Staubli VAL3: calcTool4p7En.pjx

--- calcTool4p7En.pjx ---
Parameters version=s7.3.1 stackSize=5000 millimeterUnit=true
Program file=aMainTcp.pgx
Program file=aTcp.pgx
Program file=buildTool.pgx
Program file=calculation.pgx
Program file=description.pgx
Program file=example.pgx
Program file=language.pgx
Program file=readme.pgx
Program file=splitUp.pgx
Program file=start.pgx
Program file=stop.pgx
Program file=teachPoints.pgx
Program file=usrButtonTxt.pgx
Program file=valSetBack.pgx
Data file=calcTool4p7En.dtx

--- calcTool4p7En.dtx ---
bool bAbort = true
num nLangSet = 100
num nS1[4]
num nS2[4]
num nS3[4]
num nS4[4]
num nScX
num nScY
num nScZ
num nToolX = 192.690167
num nToolY = -28.471807
num nToolZ = 149.691768
num nXPosButTxt[9]
  [2] = 5
  [3] = 10
  [4] = 15
  [5] = 20
  [6] = 25
  [7] = 30
  [8] = 35
num nYPosButTxt = 13
pointRx pTempS[5]
  [0] = {fatherId=world[0]}
  [1] = {x=378.320625, y=240.768097, z=466.569838, rx=-127.167365, ry=20.154779, rz=59.793558, shoulder=lefty, elbow=epositive, wrist=wpositive, fatherId=world[0]}
  [2] = {x=378.320625, y=240.768097, z=466.569838, rx=-127.167365, ry=20.154779, rz=59.793558, shoulder=lefty, elbow=epositive, wrist=wpositive, fatherId=world[0]}
  [3] = {x=378.320625, y=240.768097, z=466.569838, rx=-127.167365, ry=20.154779, rz=59.793558, shoulder=lefty, elbow=epositive, wrist=wpositive, fatherId=world[0]}
  [4] = {x=378.320625, y=240.768097, z=466.569838, rx=-127.167365, ry=20.154779, rz=59.793558, shoulder=lefty, elbow=epositive, wrist=wpositive, fatherId=world[0]}
string sUsrMess[140]
  [0] = "Please select a Language"
  [1] = "Programm zur Toolberechnung"
  [2] = "Dieses Prog. errechnet anhand 4 POINTS,"
  [3] = "die kugelfoermig um einen gemeinsamen"
  [4] = "Mittelpkt angeordnet sind,die X, Y und"
  [5] = "Z-Werte des akt. Tools. Diese Points"
  [6] = "muessen geometrisch unabhaengig sein."
  [7] = "D.h. sie duerfen nicht in EINER"
  [8] = "gemeinsamen Ebene liegen !!!"
  [9] = "Teachen der Locations !"
  [10] = "Punkt aufnehmen "
  [11] = "Aufnahme des "
  [12] = ".Punkts"
  [13] = "-Here- druecken um Punkt zu speichern"
  [14] = "ABBRUCH"
  [15] = "VORGANG ABGEBROCHEN !!!"
  [16] = ".Punkt aufgenommen !!!"
  [17] = "Mitte"
  [18] = "gemittelt"
  [19] = "Gemitteltes Tool sofort setzten ?"
  [20] = "TOOL NICHT GESETZT !!!"
  [21] = "TOOL GESETZT !!!"
  [22] = "Abbrechen       "
  [23] = "Wollen Sie fortfahren ? "
  [24] = " JA"
  [25] = "NEIN"
  [26] = "Here"
  [27] = "Ergebnis der Toolberechnung"
  [28] = "Tool-X"
  [29] = "Tool-Y"
  [30] = "Tool-Z"
  [31] = "Gemitteltes Tool => TRSF user_tool"
  [32] = "Division durch 0 nicht moeglich !!!"
  [101] = "Program for ToolCalculation"
  [102] = "Program to calculate the Center of a"
  [103] = "Sphere thoughout 4 POINTS which are"
  [104] = "on the surface of his Sphere. The X-,"
  [105] = "Y- and Z-Toolval. will be calcutated."
  [106] = "These POINTS have to be geometricly"
  [107] = "independant=>POINTS don't have to be"
  [108] = "located in ONE plane!!!"
  [109] = "Teaching of Locations !"
  [110] = "Teaching Location"
  [111] = "Teaching of "
  [112] = ".Point"
  [113] = "To teach the Point press - Here -"
  [114] = "ABORT"
  [115] = "PROGRAM ABORTED !!!"
  [116] = ".Point teached !!!"
  [117] = "Center"
  [118] = "average"
  [119] = "Do you want to SET average Tool now ?"
  [120] = "TOOL NOT SET !!!"
  [121] = "TOOL SET !!!"
  [122] = "Abort"
  [123] = "Do you want to continue ?"
  [124] = "YES"
  [125] = " NO"
  [126] = "Here"
  [127] = "Result of the Toolcalculation"
  [128] = "Tool-X"
  [129] = "Tool-Y"
  [130] = "Tool-Z"
  [131] = "Average Tool => TRSF user_tool"
  [132] = "Division though 0 is not possible !!!"
trsf trCenter
trsf trSphere[4]
trsf trTempTool[4]
public trsf trUserTool

--- aMainTcp.pgx ---
public program aMainTcp(num x_nUserLanguage)
  local bool l_bOk
begin
  //-----------------------------------------------------------------------
  //Header begin
  //Description of program
  //  This program creates your tool from 4 different taught positions.
  //  A wizard will guide you through the steps.
  //
  //Input parameters
  //  num x_nUserLanguage :
  //    role : defines the language of GUI (Graphical User Interface) messages
  //    possible values : 1 or 2 : 1 => Deutsch, 2 => English
  //
  //History
  //  Creation : 07-04-08 - f.Rob
  //Header end
  //-----------------------------------------------------------------------

  //Initializing all parameters (trsf, point...)
  call valSetBack()

  //Displays user title depending on the language defined
  title(sUsrMess[1+nLangSet])
  //Displays user instructions
  call description(l_bOk)
  //-> First program for teach the points, after program for calculate sphere,
  //after calculation of the tool components
  if l_bOk==true
    call teachPoints()
    call splitUp(pTempS[1],pTempS[2],pTempS[3],pTempS[4])
    call calculation(nS1[1],nS2[1],nS3[1],nS4[1],nS1[2],nS2[2],nS3[2],nS4[2],nS1[3],nS2[3],nS3[3],nS4[3])
    //Test to know if the tool calculation is correct
    //If the tool calculation is not correct (bAbort true) displays messages indicating a problem
    if bAbort
      cls()
      title("")
      gotoxy(1,6)
      putln(sUsrMess[15+nLangSet])
      put(sUsrMess[32+nLangSet])
      delay(2)
    else
      call buildTool()
    endIf
  else
    cls()
    title("")
    gotoxy(1,6)
    put(sUsrMess[15+nLangSet])
    delay(2)
  endIf
  cls()
  title("")
end

--- aTcp.pgx ---
public program aTcp(point x_pUserTcp1, point x_pUserTcp2, point x_pUserTcp3, point x_pUserTcp4, bool& x_bCalcOk[], trsf& x_trUserTool[])
begin
  //-----------------------------------------------------------------------
  //Header begin
  //Description of program
  //  Same as aMainTcp except the points need to be already taught (no wizard)
  //  Caution : Defines only the X, Y, Z components of the TCP trsf
  //
  //Input parameters
  //  point x_pUserTcp1 to x_pUserTcp4
  //    role : 4 points used to calculates the TCP
  //    possible values : not applicable (taught points)
  //
  //Output parameters
  //  bool x_bCalcOk
  //    role : set to false if there is an error of calulation and true otherwise
  //  trsf x_trUserTool
  //    role : Contains settings tool (X, Y, Z)
  //History
  //  Creation : 07-04-08 - f.Rob
  //Header end
  //-----------------------------------------------------------------------

  //Initializing all parameters (trsf, point...)
  call valSetBack()

  call splitUp(x_pUserTcp1,x_pUserTcp2,x_pUserTcp3,x_pUserTcp4)
  call calculation(nS1[1],nS2[1],nS3[1],nS4[1],nS1[2],nS2[2],nS3[2],nS4[2],nS1[3],nS2[3],nS3[3],nS4[3])
  //If the tool calculation is not correct -> bAbort true
  x_bCalcOk=!bAbort
  if bAbort
    call valSetBack()
    x_trUserTool={0,0,0,0,0,0}
  else
    x_trUserTool={nToolX,nToolY,nToolZ,0,0,0}
  endIf
end

--- buildTool.pgx ---
program buildTool()
  local num l_nI
begin
  //-----------------------------------------------------------------------
  //Header begin
  //Description of program
  //  This program filled fields X, Y, Z of trUserTool
  //
  //Traceability
  //  Creation : 07-04-08 - f.Rob
  //Header end
  //-----------------------------------------------------------------------

  userPage()
  cls()
  title(sUsrMess[27+nLangSet])
  gotoxy(1,1)
  put(sUsrMess[27+nLangSet]+":")
  gotoxy(0,3)
  //Displays a recapitulation of the 4 learning points and the components of the tool
  for l_nI=1 to 4
    put("Tool "+toString("1",l_nI)+":")
    gotoxy(8,2+l_nI)
    put("X="+toString("3.3",trTempTool[l_nI-1].x))
    gotoxy(19,2+l_nI)
    put("Y="+toString("3.3",trTempTool[l_nI-1].y))
    gotoxy(30,2+l_nI)
    putln("Z="+toString("3.3",trTempTool[l_nI-1].z))
  endFor
  gotoxy(4,8)
  put(sUsrMess[28+nLangSet]+" "+sUsrMess[18+nLangSet]+"= ")
  put(toString("3.3",nToolX))
  gotoxy(4,9)
  put(sUsrMess[29+nLangSet]+" "+sUsrMess[18+nLangSet]+"= ")
  put(toString("3.3",nToolY))
  gotoxy(4,10)
  put(sUsrMess[30+nLangSet]+" "+sUsrMess[18+nLangSet]+"= ")
  put(toString("3.3",nToolZ))
  gotoxy(2,12)
  put(sUsrMess[31+nLangSet])
  call usrButtonTxt(8,"  OK")
  wait((get()-270)==8)
  trUserTool={nToolX,nToolY,nToolZ,0,0,0}
end

--- calculation.pgx ---
program calculation(num x_nX1, num x_nX2, num x_nX3, num x_nX4, num x_nY1, num x_nY2, num x_nY3, num x_nY4, num x_nZ1, num x_nZ2, num x_nZ3, num x_nZ4)
  local num l_nTemp
  local num l_nI
  local num l_nGesamtX
  local num l_nGesamtY
  local num l_nGesamtZ
begin
  //-----------------------------------------------------------------------
  //Header begin
  //Description of program
  //  This program calculates the tool to find the X, Y, Z components
  //
  //Input parameters
  //  num x_nX1 to x_nX4
  //  num x_nY1 to x_nY4
  //  num x_nZ1 to x_nZ4
  //
  //Traceability
  //  Creation : 07-04-08 - f.Rob
  //Header end
  //-----------------------------------------------------------------------

  nScX=x_nY1*x_nX3*x_nX3*x_nZ2+x_nX1*x_nX1*x_nY2*x_nZ3-x_nX1*x_nX1*x_nY3*x_nZ2-x_nX2*x_nX2*x_nY1*x_nZ3
  nScX=nScX-x_nX3*x_nX3*x_nY2*x_nZ1-x_nY1*x_nY2*x_nY2*x_nZ3-x_nY1*x_nX4*x_nX4*x_nZ2+x_nY1*x_nY3*x_nY3*x_nZ2
  nScX=nScX+x_nY2*x_nZ1*x_nX4*x_nX4-x_nY2*x_nZ1*x_nY3*x_nY3-x_nX1*x_nX1*x_nY2*x_nZ4+x_nX1*x_nX1*x_nZ2*x_nY4
  nScX=nScX+x_nX2*x_nX2*x_nY1*x_nZ4-x_nX2*x_nX2*x_nZ1*x_nY4+x_nY1*x_nY1*x_nY2*x_nZ3-x_nY1*x_nY1*x_nY3*x_nZ2
  nScX=nScX+x_nY2*x_nY2*x_nZ1*x_nY3-x_nY1*x_nZ2*x_nY4*x_nY4+x_nY1*x_nZ2*x_nZ3*x_nZ3-x_nY1*x_nX3*x_nX3*x_nZ4
  nScX=nScX+x_nY1*x_nY2*x_nY2*x_nZ4+x_nY1*x_nX4*x_nX4*x_nZ3-x_nY1*x_nZ2*x_nZ2*x_nZ3+x_nY2*x_nZ1*x_nY4*x_nY4
  nScX=nScX-x_nY2*x_nZ1*x_nZ3*x_nZ3+x_nY2*x_nZ1*x_nZ1*x_nZ3+x_nZ1*x_nY3*x_nZ2*x_nZ2-x_nZ1*x_nX4*x_nX4*x_nY3
  nScX=nScX+x_nX1*x_nX1*x_nY3*x_nZ4-x_nX1*x_nX1*x_nY4*x_nZ3-x_nY1*x_nY1*x_nY2*x_nZ4+x_nY1*x_nY1*x_nZ2*x_nY4
  nScX=nScX+x_nX3*x_nX3*x_nZ1*x_nY4-x_nY2*x_nY2*x_nZ1*x_nY4-x_nZ1*x_nZ1*x_nY3*x_nZ2-x_nY1*x_nZ2*x_nZ4*x_nZ4
  nScX=nScX-x_nY1*x_nY3*x_nY3*x_nZ4+x_nY1*x_nZ2*x_nZ2*x_nZ4+x_nY1*x_nY4*x_nY4*x_nZ3+x_nY2*x_nZ1*x_nZ4*x_nZ4
  nScX=nScX-x_nY2*x_nZ1*x_nZ1*x_nZ4-x_nY2*x_nX4*x_nX4*x_nZ3-x_nZ1*x_nY3*x_nY4*x_nY4+x_nZ1*x_nY3*x_nY3*x_nY4
  nScX=nScX-x_nZ1*x_nZ2*x_nZ2*x_nY4-x_nX2*x_nX2*x_nY3*x_nZ4+x_nX2*x_nX2*x_nY4*x_nZ3+x_nY1*x_nY1*x_nY3*x_nZ4
  nScX=nScX-x_nY1*x_nY1*x_nY4*x_nZ3+x_nX3*x_nX3*x_nY2*x_nZ4-x_nX3*x_nX3*x_nZ2*x_nY4+x_nZ1*x_nZ1*x_nZ2*x_nY4
  nScX=nScX+x_nX4*x_nX4*x_nY3*x_nZ2+x_nY1*x_nZ3*x_nZ4*x_nZ4-x_nY1*x_nZ3*x_nZ3*x_nZ4+x_nY2*x_nY3*x_nY3*x_nZ4
  nScX=nScX-x_nY2*x_nY4*x_nY4*x_nZ3-x_nZ1*x_nY3*x_nZ4*x_nZ4+x_nZ1*x_nY4*x_nZ3*x_nZ3+x_nY3*x_nZ2*x_nY4*x_nY4
  nScX=nScX-x_nY2*x_nY2*x_nY3*x_nZ4+x_nY2*x_nY2*x_nY4*x_nZ3+x_nZ1*x_nZ1*x_nY3*x_nZ4-x_nZ1*x_nZ1*x_nY4*x_nZ3
  nScX=nScX-x_nY3*x_nY3*x_nZ2*x_nY4-x_nY2*x_nZ3*x_nZ4*x_nZ4+x_nY2*x_nZ3*x_nZ3*x_nZ4+x_nY3*x_nZ2*x_nZ4*x_nZ4
  nScX=nScX-x_nY3*x_nZ2*x_nZ2*x_nZ4-x_nZ2*x_nY4*x_nZ3*x_nZ3+x_nZ2*x_nZ2*x_nY4*x_nZ3+x_nX2*x_nX2*x_nZ1*x_nY3
  l_nTemp=2*x_nX1*x_nY2*x_nZ3-2*x_nX1*x_nY3*x_nZ2-2*x_nX2*x_nY1*x_nZ3+2*x_nX2*x_nZ1*x_nY3+2*x_nY1*x_nX3*x_nZ2
  l_nTemp=l_nTemp-2*x_nX3*x_nY2*x_nZ1-2*x_nX1*x_nY2*x_nZ4+2*x_nX1*x_nZ2*x_nY4+2*x_nX2*x_nY1*x_nZ4-2*x_nX2*x_nZ1*x_nY4-2*x_nY1*x_nX4*x_nZ2
  l_nTemp=l_nTemp+2*x_nY2*x_nZ1*x_nX4+2*x_nX1*x_nY3*x_nZ4-2*x_nX1*x_nY4*x_nZ3-2*x_nY1*x_nX3*x_nZ4+2*x_nY1*x_nX4*x_nZ3+2*x_nX3*x_nZ1*x_nY4
  l_nTemp=l_nTemp-2*x_nZ1*x_nX4*x_nY3-2*x_nX2*x_nY3*x_nZ4+2*x_nX2*x_nY4*x_nZ3+2*x_nX3*x_nY2*x_nZ4-2*x_nX3*x_nZ2*x_nY4-2*x_nY2*x_nX4*x_nZ3
  l_nTemp=l_nTemp+2*x_nX4*x_nY3*x_nZ2
  if abs(l_nTemp)<0.001
    nScX=9999.9999
  else
    nScX=nScX/l_nTemp
  endIf
  nScY=x_nX1*x_nX2*x_nX2*x_nZ3-x_nX1*x_nX3*x_nX3*x_nZ2+x_nX2*x_nX3*x_nX3*x_nZ1-x_nX1*x_nX1*x_nX2*x_nZ3
  nScY=nScY+x_nX1*x_nX1*x_nX3*x_nZ2-x_nX2*x_nX2*x_nX3*x_nZ1-x_nX1*x_nX2*x_nX2*x_nZ4+x_nX1*x_nY2*x_nY2*x_nZ3
  nScY=nScY+x_nX1*x_nX4*x_nX4*x_nZ2-x_nX1*x_nY3*x_nY3*x_nZ2-x_nX2*x_nZ1*x_nX4*x_nX4+x_nX2*x_nZ1*x_nY3*x_nY3
  nScY=nScY-x_nX2*x_nY1*x_nY1*x_nZ3-x_nX3*x_nY2*x_nY2*x_nZ1+x_nX1*x_nX1*x_nX2*x_nZ4-x_nX1*x_nX1*x_nX4*x_nZ2
  nScY=nScY+x_nX2*x_nX2*x_nZ1*x_nX4+x_nY1*x_nY1*x_nX3*x_nZ2+x_nX1*x_nZ2*x_nY4*x_nY4-x_nX1*x_nZ2*x_nZ3*x_nZ3
  nScY=nScY+x_nX1*x_nX3*x_nX3*x_nZ4-x_nX1*x_nY2*x_nY2*x_nZ4-x_nX1*x_nX4*x_nX4*x_nZ3+x_nX1*x_nZ2*x_nZ2*x_nZ3
  nScY=nScY-x_nX2*x_nZ1*x_nY4*x_nY4+x_nX2*x_nZ1*x_nZ3*x_nZ3+x_nX2*x_nY1*x_nY1*x_nZ4-x_nX2*x_nZ1*x_nZ1*x_nZ3
  nScY=nScY+x_nX3*x_nZ1*x_nX4*x_nX4-x_nX3*x_nZ1*x_nZ2*x_nZ2+x_nX3*x_nZ1*x_nZ1*x_nZ2-x_nX1*x_nX1*x_nX3*x_nZ4
  nScY=nScY+x_nX1*x_nX1*x_nX4*x_nZ3-x_nY1*x_nY1*x_nX4*x_nZ2-x_nX3*x_nX3*x_nZ1*x_nX4+x_nY2*x_nY2*x_nZ1*x_nX4
  nScY=nScY+x_nX1*x_nZ2*x_nZ4*x_nZ4+x_nX1*x_nY3*x_nY3*x_nZ4-x_nX1*x_nZ2*x_nZ2*x_nZ4-x_nX1*x_nY4*x_nY4*x_nZ3
  nScY=nScY-x_nX2*x_nZ1*x_nZ4*x_nZ4-x_nX2*x_nX3*x_nX3*x_nZ4+x_nX2*x_nZ1*x_nZ1*x_nZ4+x_nX2*x_nX4*x_nX4*x_nZ3
  nScY=nScY+x_nX3*x_nZ1*x_nY4*x_nY4-x_nX3*x_nX4*x_nX4*x_nZ2-x_nZ1*x_nX4*x_nY3*x_nY3+x_nZ1*x_nX4*x_nZ2*x_nZ2
  nScY=nScY+x_nX2*x_nX2*x_nX3*x_nZ4-x_nX2*x_nX2*x_nX4*x_nZ3-x_nY1*x_nY1*x_nX3*x_nZ4+x_nY1*x_nY1*x_nX4*x_nZ3
  nScY=nScY+x_nX3*x_nX3*x_nX4*x_nZ2-x_nZ1*x_nZ1*x_nX4*x_nZ2-x_nX1*x_nZ3*x_nZ4*x_nZ4+x_nX1*x_nZ3*x_nZ3*x_nZ4
  nScY=nScY-x_nX2*x_nY3*x_nY3*x_nZ4+x_nX2*x_nY4*x_nY4*x_nZ3+x_nX3*x_nZ1*x_nZ4*x_nZ4-x_nX3*x_nZ2*x_nY4*x_nY4
  nScY=nScY+x_nX3*x_nY2*x_nY2*x_nZ4-x_nX3*x_nZ1*x_nZ1*x_nZ4-x_nZ1*x_nX4*x_nZ3*x_nZ3+x_nX4*x_nY3*x_nY3*x_nZ2
  nScY=nScY-x_nY2*x_nY2*x_nX4*x_nZ3+x_nZ1*x_nZ1*x_nX4*x_nZ3+x_nX2*x_nZ3*x_nZ4*x_nZ4-x_nX2*x_nZ3*x_nZ3*x_nZ4
  nScY=nScY-x_nX3*x_nZ2*x_nZ4*x_nZ4+x_nX3*x_nZ2*x_nZ2*x_nZ4+x_nX4*x_nZ2*x_nZ3*x_nZ3-x_nX4*x_nZ2*x_nZ2*x_nZ3
  l_nTemp=2*x_nX1*x_nY2*x_nZ3-2*x_nX1*x_nY3*x_nZ2-2*x_nX2*x_nY1*x_nZ3+2*x_nX2*x_nZ1*x_nY3
  l_nTemp=l_nTemp+2*x_nY1*x_nX3*x_nZ2-2*x_nX3*x_nY2*x_nZ1-2*x_nX1*x_nY2*x_nZ4+2*x_nX1*x_nZ2*x_nY4+2*x_nX2*x_nY1*x_nZ4-2*x_nX2*x_nZ1*x_nY4
  l_nTemp=l_nTemp-2*x_nY1*x_nX4*x_nZ2+2*x_nY2*x_nZ1*x_nX4+2*x_nX1*x_nY3*x_nZ4-2*x_nX1*x_nY4*x_nZ3-2*x_nY1*x_nX3*x_nZ4+2*x_nY1*x_nX4*x_nZ3
  l_nTemp=l_nTemp+2*x_nX3*x_nZ1*x_nY4-2*x_nZ1*x_nX4*x_nY3-2*x_nX2*x_nY3*x_nZ4+2*x_nX2*x_nY4*x_nZ3+2*x_nX3*x_nY2*x_nZ4-2*x_nX3*x_nZ2*x_nY4
  l_nTemp=l_nTemp-2*x_nY2*x_nX4*x_nZ3+2*x_nX4*x_nY3*x_nZ2
  if abs(l_nTemp)<0.001
    nScY=9999.9999
  else
    nScY=nScY/l_nTemp
  endIf
  nScZ=x_nX1*x_nX3*x_nX3*x_nY2-x_nX1*x_nX2*x_nX2*x_nY3-x_nX2*x_nY1*x_nX3*x_nX3+x_nX1*x_nX1*x_nX2*x_nY3
  nScZ=nScZ-x_nX1*x_nX1*x_nX3*x_nY2+x_nX2*x_nX2*x_nY1*x_nX3-x_nX1*x_nY2*x_nX4*x_nX4+x_nX1*x_nY2*x_nY3*x_nY3
  nScZ=nScZ+x_nX1*x_nX2*x_nX2*x_nY4-x_nX1*x_nY2*x_nY2*x_nY3+x_nX2*x_nY1*x_nX4*x_nX4-x_nX2*x_nY1*x_nY3*x_nY3
  nScZ=nScZ+x_nX2*x_nY1*x_nY1*x_nY3+x_nY1*x_nX3*x_nY2*x_nY2-x_nX1*x_nX1*x_nX2*x_nY4+x_nX1*x_nX1*x_nY2*x_nX4
  nScZ=nScZ-x_nX2*x_nX2*x_nY1*x_nX4-x_nY1*x_nY1*x_nX3*x_nY2-x_nX1*x_nY2*x_nY4*x_nY4+x_nX1*x_nY2*x_nZ3*x_nZ3
  nScZ=nScZ-x_nX1*x_nY3*x_nZ2*x_nZ2-x_nX1*x_nX3*x_nX3*x_nY4+x_nX1*x_nY2*x_nY2*x_nY4+x_nX1*x_nX4*x_nX4*x_nY3
  nScZ=nScZ+x_nX2*x_nY1*x_nY4*x_nY4-x_nX2*x_nY1*x_nZ3*x_nZ3-x_nX2*x_nY1*x_nY1*x_nY4+x_nX2*x_nZ1*x_nZ1*x_nY3
  nScZ=nScZ-x_nY1*x_nX3*x_nX4*x_nX4+x_nY1*x_nX3*x_nZ2*x_nZ2+x_nY1*x_nX3*x_nX3*x_nX4-x_nY1*x_nY2*x_nY2*x_nX4
  nScZ=nScZ-x_nX3*x_nY2*x_nZ1*x_nZ1+x_nX1*x_nX1*x_nX3*x_nY4-x_nX1*x_nX1*x_nX4*x_nY3+x_nY1*x_nY1*x_nY2*x_nX4
  nScZ=nScZ-x_nX1*x_nY2*x_nZ4*x_nZ4+x_nX1*x_nY3*x_nY4*x_nY4-x_nX1*x_nY3*x_nY3*x_nY4+x_nX1*x_nZ2*x_nZ2*x_nY4
  nScZ=nScZ+x_nX2*x_nY1*x_nZ4*x_nZ4+x_nX2*x_nX3*x_nX3*x_nY4-x_nX2*x_nZ1*x_nZ1*x_nY4-x_nX2*x_nX4*x_nX4*x_nY3
  nScZ=nScZ-x_nY1*x_nX3*x_nY4*x_nY4+x_nY1*x_nX4*x_nY3*x_nY3-x_nY1*x_nX4*x_nZ2*x_nZ2+x_nX3*x_nY2*x_nX4*x_nX4
  nScZ=nScZ+x_nY2*x_nZ1*x_nZ1*x_nX4-x_nX2*x_nX2*x_nX3*x_nY4+x_nX2*x_nX2*x_nX4*x_nY3+x_nY1*x_nY1*x_nX3*x_nY4
  nScZ=nScZ-x_nY1*x_nY1*x_nX4*x_nY3-x_nX3*x_nX3*x_nY2*x_nX4+x_nX1*x_nY3*x_nZ4*x_nZ4-x_nX1*x_nY4*x_nZ3*x_nZ3
  nScZ=nScZ-x_nX2*x_nY3*x_nY4*x_nY4+x_nX2*x_nY3*x_nY3*x_nY4-x_nY1*x_nX3*x_nZ4*x_nZ4+x_nY1*x_nX4*x_nZ3*x_nZ3
  nScZ=nScZ+x_nX3*x_nY2*x_nY4*x_nY4-x_nX3*x_nY2*x_nY2*x_nY4+x_nX3*x_nZ1*x_nZ1*x_nY4-x_nY2*x_nX4*x_nY3*x_nY3
  nScZ=nScZ+x_nY2*x_nY2*x_nX4*x_nY3-x_nZ1*x_nZ1*x_nX4*x_nY3-x_nX2*x_nY3*x_nZ4*x_nZ4+x_nX2*x_nY4*x_nZ3*x_nZ3
  nScZ=nScZ+x_nX3*x_nY2*x_nZ4*x_nZ4-x_nX3*x_nZ2*x_nZ2*x_nY4-x_nY2*x_nX4*x_nZ3*x_nZ3+x_nX4*x_nY3*x_nZ2*x_nZ2
  l_nTemp=2*x_nX1*x_nY2*x_nZ3-2*x_nX1*x_nY3*x_nZ2-2*x_nX2*x_nY1*x_nZ3+2*x_nX2*x_nZ1*x_nY3+2*x_nY1*x_nX3*x_nZ2-2*x_nX3*x_nY2*x_nZ1
  l_nTemp=l_nTemp-2*x_nX1*x_nY2*x_nZ4+2*x_nX1*x_nZ2*x_nY4+2*x_nX2*x_nY1*x_nZ4-2*x_nX2*x_nZ1*x_nY4-2*x_nY1*x_nX4*x_nZ2+2*x_nY2*x_nZ1*x_nX4
  l_nTemp=l_nTemp+2*x_nX1*x_nY3*x_nZ4-2*x_nX1*x_nY4*x_nZ3-2*x_nY1*x_nX3*x_nZ4+2*x_nY1*x_nX4*x_nZ3+2*x_nX3*x_nZ1*x_nY4-2*x_nZ1*x_nX4*x_nY3
  l_nTemp=l_nTemp-2*x_nX2*x_nY3*x_nZ4+2*x_nX2*x_nY4*x_nZ3+2*x_nX3*x_nY2*x_nZ4-2*x_nX3*x_nZ2*x_nY4-2*x_nY2*x_nX4*x_nZ3+2*x_nX4*x_nY3*x_nZ2
  if abs(l_nTemp)<0.001
    nScZ=9999.9999
  else
    nScZ=nScZ/l_nTemp
  endIf
  if ((nScX==9999.9999) or (nScY==9999.9999) or (nScZ==9999.9999))
    bAbort=true
    call valSetBack()
  else
    bAbort=false
    //Theoretical Center of Sphere
    trCenter={nScX,nScY,nScZ,0,0,0}
    //Inverse sphere * center
    for l_nI=0 to 3
      trTempTool[l_nI]=!trSphere[l_nI]*trCenter
    endFor
    l_nGesamtX=0
    l_nGesamtY=0
    l_nGesamtZ=0
    for l_nI=0 to 3
      l_nGesamtX=l_nGesamtX+trTempTool[l_nI].x
      l_nGesamtY=l_nGesamtY+trTempTool[l_nI].y
      l_nGesamtZ=l_nGesamtZ+trTempTool[l_nI].z
    endFor
    nToolX=l_nGesamtX/4
    nToolY=l_nGesamtY/4
    nToolZ=l_nGesamtZ/4
  endIf
end

--- description.pgx ---
program description(bool& x_bOk[])
  local num l_nI
  local num l_nWhich
begin
  //-----------------------------------------------------------------------
  //Header begin
  //Description of program
  //  This program lets you choose the keys to display
  //
  //Input parameters
  //  bool x_bOK
  //    role : User's choice: continue or stop the program
  //    possible values : 0 or 1 : 0 => Stop program, 1 => continue
  //
  //Traceability
  //  Creation : 07-04-08 - f.Rob
  //Header end
  //-----------------------------------------------------------------------

  x_bOk=false
  userPage()
  gotoxy(0,1)
  //Displays user instructions depending on the language defined
  for l_nI=(1+nLangSet) to (8+nLangSet)
    putln(sUsrMess[l_nI])
  endFor
  gotoxy(8,10)
  put(sUsrMess[23+nLangSet])
  //Functions to display navigation keys (F1 through F8)(here F3 and F6 with messages "YES" or "NO")
  call usrButtonTxt(3,sUsrMess[24+nLangSet])
  call usrButtonTxt(6,sUsrMess[25+nLangSet])
  //Waiting user choice: F3 or F6
  //F3=3 The user wants to continue
  //F6=6 The user wants to quit
  do
    l_nWhich=(get()-270)
  until ((l_nWhich==3) or (l_nWhich==6))
  //if the user wants to continue (he press F3) x_bOk passes true
  if l_nWhich==3
    x_bOk=true
  endIf
end

--- example.pgx ---
program example()
  local num l_nLanguage
begin
  //-----------------------------------------------------------------------
  //Header begin
  //Description of program
  //  This is an example for use this library.
  //  This program run differents sub-programs :
  //  - language() for choose the language : "English or "Deutsch"
  //  - aMainTcp() for calculates the tool transformation : a wizard will
  //  guide you thtough the steps.
  //
  //Traceability
  //  Creation : 08-04-08 - f.Rob
  //Header end
  //-----------------------------------------------------------------------

  call language()
  call aMainTcp(nLangSet)
end

--- language.pgx ---
public program language()
  local num l_nWhich
begin
  //-----------------------------------------------------------------------
  //Header begin
  //Description of program
  //  This program lets you choose the language : English or Deutsch
  //
  //Traceability
  //  Creation : 07-04-08 - f.Rob
  //Header end
  //-----------------------------------------------------------------------
  userPage()
  cls()
  gotoxy(5,5)
  putln(sUsrMess[101])
  gotoxy(7,10)
  put(sUsrMess[0])
  //Functions to display navigation keys (F1 through F8)
  //(here F3 and F6 with messages "Germ" or "Engl")
  call usrButtonTxt(3,"Germ")
  call usrButtonTxt(6,"Engl")
  //Waiting user choice 3 (F3) or 6 (F6)
  do
    l_nWhich=(get()-270)
  until ((l_nWhich==3) or (l_nWhich==6))
  //User choice : 3 (F3)=> Deutsch, 6 (F6)=> English
  switch l_nWhich
    case 3
      nLangSet=0
    break
    case 6
      nLangSet=100
    break
  endSwitch
  cls()
  userPage()
  gotoxy(0,13)
  put("                                       ")
end

--- readme.pgx ---
program readme()
begin
  //Title: Calculates a tool transformation
  //
  //General description :
  //  This library calculates a tool transformation
  //  without the need to a teach reference point.
  //  Jog robot to a single location with 4 different orientations
  //  with the tool you want to teach mounted on the robot.
  //  Select tool "flange" when teaching the points.
  //  Caution : Defines only the X, Y, Z components of the TCP's trsf
  //
  //Hardware required :
  //  - Robot system    : any 6 axis Staubli robot
  //  - Peripherals     : no peripherals required
  //
  //VAL3 options :
  //  - VAL3 version    : 7.3
  //  - VAL3 licenses   : no licenses required
  //  - VAL3 add-ons    : none
  //
  //Library version     : 7.3.1.0
  //
  //Public variables    : none
  //
  //Included libraries  : none
  //
  //Miscellaneous       : switched to version 7, IO library removed, no other modification - T.Caille 04/2012
  //
  //Keywords            : calculates, calcul, tool, outil, 4 different orientations, 4 orientations differentes, point, components, composantes
end

--- splitUp.pgx ---
program splitUp(point x_pSphere1, point x_pSphere2, point x_pSphere3, point x_pSphere4)
begin
  //-----------------------------------------------------------------------
  //Header begin
  //Description of program
  //  This program calculates the sphere.
  //
  //Input parameters
  //  point x_pSphere1 to point x_pSphere4 :
  //
  //Traceability
  //  Creation : 07-04-08 - f.Rob
  //Header end
  //-----------------------------------------------------------------------

  trSphere[0]=x_pSphere1.trsf
  trSphere[1]=x_pSphere2.trsf
  trSphere[2]=x_pSphere3.trsf
  trSphere[3]=x_pSphere4.trsf
  nS1[1]=trSphere[0].x
  nS1[2]=trSphere[0].y
  nS1[3]=trSphere[0].z
  nS2[1]=trSphere[1].x
  nS2[2]=trSphere[1].y
  nS2[3]=trSphere[1].z
  nS3[1]=trSphere[2].x
  nS3[2]=trSphere[2].y
  nS3[3]=trSphere[2].z
  nS4[1]=trSphere[3].x
  nS4[2]=trSphere[3].y
  nS4[3]=trSphere[3].z
end

--- stop.pgx ---
program stop()
begin
  popUpMsg("Press CS8 to get back to Main Menue")
  resetMotion()
end

--- teachPoints.pgx ---
program teachPoints()
  local num l_nI
  local num l_nWhich
begin
  //-----------------------------------------------------------------------
  //Header begin
  //Description of program
  //  This program allows you to teach 4 points
  //
  //Traceability
  //  Creation : 07-04-08 - f.Rob
  //Header end
  //-----------------------------------------------------------------------

  userPage()
  cls()
  gotoxy(2,2)
  put(sUsrMess[9+nLangSet])
  gotoxy(1,9)
  put(sUsrMess[13+nLangSet])
  //Function to display navigation keys (F1 through F8) (here F4 with message "Here")
  call usrButtonTxt(4,sUsrMess[26+nLangSet])
  //Loop to remember 4 points
  for l_nI=1 to 4
    gotoxy(2,4)
    //Displays point during the apprenticeship (ex: Teaching of 2.Point)
    putln(sUsrMess[11+nLangSet]+toString("1",l_nI)+sUsrMess[12+nLangSet])
    putln("")
    put("----------------------------------------")
    //Waiting pressing 4 (F4 key) for memorize the point
    wait((get()-270)==4)
    pTempS[l_nI]=here(flange,world)
  endFor
end

--- usrButtonTxt.pgx ---
program usrButtonTxt(num x_nWhichButton, string x_sButtonTxt)
begin
  //-----------------------------------------------------------------------
  //Header begin
  //Description of program
  //  This program lets you choose the button to display
  //
  //Input parameters
  //  num x_nWhichButton :
  //    role : choice of the navigation key
  //    possible values : 1 to 8 (F1 to F8)
  //
  //  string x_sButtonTxt :
  //    role : Displays desired text
  //
  //Traceability
  //  Creation : 07-04-08 - f.Rob
  //Header end
  //-----------------------------------------------------------------------

  //Position cursor X, Y
  gotoxy(nXPosButTxt[x_nWhichButton],nYPosButTxt)
  //Displays Text
  put(left(x_sButtonTxt,4))
  //Erases contents of  text button parameters
  x_sButtonTxt=" "
end

--- valSetBack.pgx ---
program valSetBack()
  local num l_nI
begin
  //-----------------------------------------------------------------------
  //Header begin
  //Description of program
  //  This program initializes various variables
  //
  //Traceability
  //  Creation : 07-04-08 - f.Rob
  //Header end
  //-----------------------------------------------------------------------

  for l_nI=0 to 3
    trSphere[l_nI]={0,0,0,0,0,0}
  endFor
  for l_nI=0 to 4
    pTempS[0].trsf=trSphere[0]
  endFor
  for l_nI=0 to 3
    trTempTool[l_nI]={0,0,0,0,0,0}
    nS1[l_nI]=nS2[l_nI]=nS3[l_nI]=nS4[l_nI]=0
  endFor
  nScX=nScY=nScZ=0
  trCenter={0,0,0,0,0,0}
  trUserTool={0,0,0,0,0,0}
end
